FUNCTION_BLOCK PUBLIC BoolIn IMPLEMENTS I_StepCondition
VAR_INPUT
END_VAR
VAR_OUTPUT
END_VAR
VAR
	bValue AT%I* : BOOL;
END_VAR

{warning 'Eigenschaftenimplementierung hinzufügen'}
PROPERTY getValue : BOOL
GET
getValue := bValue;
END_GET
END_PROPERTY

{warning 'Eigenschaftenimplementierung hinzufügen'}
PROPERTY setValue : BOOL
SET
bValue := setValue;
END_SET
END_PROPERTY

END_FUNCTION_BLOCK

(* stored: Version 1.1.0.1, ProductVersion 3.1.4024.0
   POU BoolIn: Id {370a6c08-2d5a-402b-b600-192f1fdc1dc6}, SpecialFunc None
   Property getValue: Id {641c2af3-70fb-41ab-be46-84f24b7f90b0}
   Get Get: Id {7ebe42a3-3ad0-437c-82d6-968da80e6195}
   Property setValue: Id {89adadce-2c51-491c-a739-6235884b2a94}
   Set Set: Id {08200bd5-86b2-47c7-b485-02f152ca4088} *)
